Fanuc KAREL source: kt00378.KL

-- PROVISIONAL review KL for V1013-1; original PC SHA256 f520bf88504ae37de7370e0496638cfb5b2dc309d1339027726f737f47f58d53
-- Incomplete behavior may be omitted. Consult companion uncertainty JSON. Do not deploy.
PROGRAM KT00378
%NOLOCKGROUP
VAR
  OUT : BOOLEAN
-- UNRESOLVED_DECL Y1 type=002018
-- UNRESOLVED_DECL H2 type=002017
BEGIN
  -- UNRESOLVED_PC offsets 5-19; opcodes 2E,22,9D,33,B2
  -- UNRESOLVED_PC offsets 24-38; opcodes 2E,22,9D,33,B4
  -- UNRESOLVED_PC offsets 43-68; opcodes 22,9D,33,B1,22,9D,33,B3,5A,23
  -- UNRESOLVED_PC offsets 73-77; opcodes 7F
END KT00378
